// TIA Portal V17 export
// export: Created 2023-04-03T06:31:30.3814142Z, ExportSetting WithDefaults, DisplayName Totally Integrated Automation Portal, DisplayVersion V17 Update 4, DisplayName TIA Portal Openness, DisplayVersion V17 Update 4, DisplayName TIA Portal Version Control Interface, DisplayVersion V17, DisplayName STEP 7 Professional, DisplayVersion V17 Update 4, DisplayName STEP 7 Safety, DisplayVersion V17, DisplayName WinCC Professional, DisplayVersion V17 Update 4
DATA_BLOCK "SS"   // DB101
{ S7_Optimized_Access := 'TRUE' }
VERSION : 0.1
// stored: AutoNumber false, DBAccessibleFromOPCUA true, DBAccessibleFromWebserver true, IsOnlyStoredInLoadMemory false, IsRetainMemResEnabled false, IsWriteProtectedInAS false, MemoryReserve 100
   VAR
      xFltSt : Bool;
      xSs1FltSt : Bool;
      xSs2FltSt : Bool;
      xAlmSt : Bool;
      XWarSt : Bool;   // Warning status
      wAlm1 : Word;
      wAlm2 : Word;
      wAlm3 : Word;
      wAlm4 : Word;
      wAlm5 : Word;
      wWarn1 : Word;
      wWarn2 : Word;
      wWarn3 : Word;
      wWarn4 : Word;
      wWarn5 : Word;
   END_VAR
BEGIN
END_DATA_BLOCK
